FUNCTION_BLOCK GET_PLANE_LOWEST_POINT (* Get plane lowest point *)
  (* Standard: 61499-2 *)
  (* Version 1.0, 05-07-12, GASR, Universidade do Estado de Santa Catarina *)
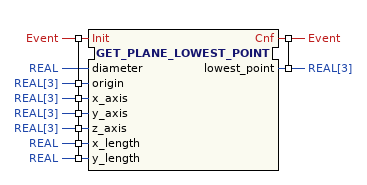
  EVENT_INPUT
    Init WITH origin, x_axis, y_axis, z_axis, x_length, y_length;
  END_EVENT
  EVENT_OUTPUT
    Cnf WITH lowest_point;
  END_EVENT
  VAR_INPUT
    diameter : REAL; (* Tool diameter *)
    origin : ARRAY [0..2] OF REAL; (* Plane origin point *)
    x_axis : ARRAY [0..2] OF REAL; (* reference axis *)
    y_axis : ARRAY [0..2] OF REAL; (* OP axis *)
    z_axis : ARRAY [0..2] OF REAL; (* normal vector *)
    x_length : REAL;
    y_length : REAL;
  END_VAR
  VAR_OUTPUT
    lowest_point : ARRAY [0..2] OF REAL;
  END_VAR
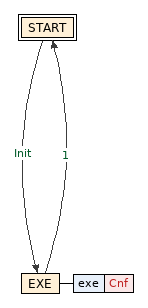
  EC_STATES
    START;
    EXE : exe -> Cnf;
  END_STATES
  EC_TRANSITIONS
    START TO EXE := Init;
    EXE TO START := 1;
  END_TRANSITIONS
  ALGORITHM exe IN Lua:
x_length = x_length - diameter
y_length = y_length - diameter
if(( x_axis[1] == 0 ) and ( x_axis[2] == 0 ) and ( x_axis[3] == 0 )) then
    x_axis = { ((y_axis[2]*z_axis[3]) - (z_axis[2]*y_axis[3])),
                    ((y_axis[3]*z_axis[1]) - (z_axis[3]*y_axis[1])),
                    ((y_axis[1]*z_axis[2]) - (z_axis[1]*y_axis[2])) }
elseif(( y_axis[1] == 0 ) and ( y_axis[2] == 0 ) and ( y_axis[3] == 0 )) then
    y_axis = { ((z_axis[2]*x_axis[3]) - (x_axis[2]*z_axis[3])),
                    ((z_axis[3]*x_axis[1]) - (x_axis[3]*z_axis[1])),
                    ((z_axis[1]*x_axis[2]) - (x_axis[1]*z_axis[2])) }
elseif(( z_axis[1] == 0 ) and ( z_axis[2] == 0 ) and ( z_axis[3] == 0 )) then
    z_axis = { ((x_axis[2]*y_axis[3]) - (y_axis[2]*x_axis[3])),
                    ((x_axis[3]*y_axis[1]) - (y_axis[3]*x_axis[1])),
                    ((x_axis[1]*y_axis[2]) - (y_axis[1]*x_axis[2])) }
end
local points = { { origin[1], origin[2], origin[3] } }
local opp_point = { ( origin[1] + x_axis[1]*x_length + y_axis[1]*y_length ),
                    ( origin[2] + x_axis[2]*x_length + y_axis[2]*y_length ), origin[3] }
local t, w
if( y_axis[1] == 0 ) then
    t = ( opp_point[1]/x_axis[1] - origin[1] )
    w = ( opp_point[2] - origin[2] - x_axis[2]*t )/y_axis[2]
elseif( x_axis[1] == 0 ) then
    w = ( opp_point[1]/y_axis[1] - origin[2] )
    t = ( opp_point[2] - origin[2] - y_axis[2]*w )/y_axis[2]
else
    t = ( ( opp_point[2] - y_axis[2]*opp_point[1]/y_axis[1] + y_axis[2]*origin[1]/y_axis[1] - origin[2] )/( x_axis[2] - y_axis[2]*x_axis[2]/y_axis[1] ) )
    w = ( opp_point[1] - origin[1] - x_axis[1]*t )/y_axis[1]
end
opp_point[3] = ( x_axis[3]*t + y_axis[3]*w + origin[3] )
points[2] = { opp_point[1], opp_point[2], opp_point[3] }
points[3] = { opp_point[1], origin[2], x_axis[3]*t + origin[3] }
points[4] = { origin[1], opp_point[2], y_axis[3]*w + origin[3] }
if(( points[2][3] >= points[1][3] ) and ( points[3][3] >= points[1][3] ) and ( points[4][3] >= points[1][3] )) then
    lowest_point = { points[1][1], points[1][2], points[1][3] }
elseif(( points[1][3] >= points[2][3] ) and ( points[3][3] >= points[2][3] ) and ( points[4][3] >= points[2][3] )) then
    lowest_point = { points[2][1], points[2][2], points[2][3] }
elseif(( points[1][3] >= points[3][3] ) and ( points[2][3] >= points[3][3] ) and ( points[4][3] >= points[3][3] )) then
    lowest_point = { points[3][1], points[3][2], points[3][3] }
else
    lowest_point = { points[4][1], points[4][2], points[4][3] }
end
print( '\nlowest_points', lowest_point[3], points[1][3], points[2][3], points[3][3], points[4][3], '\n' )
  END_ALGORITHM
END_FUNCTION_BLOCK
